TYPE TelemetryIOStatuses :
STRUCT
	///Is the I/O in a healthy state?
	healthStatus: HealthStatus;
END_STRUCT
END_TYPE

(* stored: Version 1.1.0.1, ProductVersion 3.1.4019.2
   DUT TelemetryIOStatuses: Id {2baece0b-2875-4d72-81f6-486a3013b3da} *)
